TYPE ST_OPC_UA_Node :
STRUCT
	NodeID				: ST_UANodeID;
	NodeHdl				: DWORD;
	SizeOfDataType		: UDINT;
	NodeAddInfo			: ST_UANodeAdditionalInfo;
	TargetVar			: POINTER TO BOOL;
END_STRUCT
END_TYPE

(* stored: Version 1.1.0.1, ProductVersion 3.1.4024.9
   DUT ST_OPC_UA_Node: Id {e5d3d981-1f38-4aa1-a57f-322359324821} *)
